// TwinCAT 3 PLC project Untitled1
// ProgramVersion: 3.1.4024.0
// libraries:
//   Tc2_Standard, * (Beckhoff Automation GmbH)
//   Tc2_System, * (Beckhoff Automation GmbH)
//   Tc3_Module, * (Beckhoff Automation GmbH)
//   VisuSymbols,3.5.10.0,System
// project tree:
//   / GlobalTextList.TcGTLO, PlcTask.TcTTO, Visualization Manager.TcVMO (not stored), Visualization.TcVIS
//   GVLs/ GVL.TcGVL
//   POUs/ MAIN.TcPOU, VeranderLicht.TcPOU, VerkeersLichtL.TcPOU, VerkeersLichtR.TcPOU, VerkeerslichtStatus.TcTLEO
// real-time tasks:
//   TASK PlcTask: cycle T#10ms, priority 20, ADS port 350
//   TASK Task 4: cycle T#10ms, priority 1, ADS port 351

CONFIGURATION Untitled1
    RESOURCE PLC ON TwinCAT3
        TASK PlcTask(INTERVAL := T#10ms, PRIORITY := 20);
        PROGRAM MAIN WITH PlcTask : MAIN;
    END_RESOURCE
END_CONFIGURATION

// ---- POUs/VerkeerslichtStatus.TcTLEO
{attribute 'qualified_only'}
{attribute 'strict'}
TYPE VerkeerslichtStatus :
(
	Rood := 0,    // 0
    Geel := 1,    // 1
    Groen := 2    // 2
);
END_TYPE

// ---- GVLs/GVL.TcGVL
{attribute 'qualified_only'}
VAR_GLOBAL
	GroenR : BOOL; 
	GeelR : BOOL;
	RoodR: BOOL;
	GroenL : BOOL;
	GeelL : BOOL;
	RoodL: BOOL;
	
	LichtStatusR: INT := 0; // 0 = Rood, 1 = Groen, 2 = Oranje
	LichtStatusL: INT := 0; // 0 = Rood, 1 = Groen, 2 = Oranje
	
	AutoR : BOOL; // Auto komt van Rechts
	AutoL : BOOL; // Auto komt van Links
	
	TijdGroen : TIME := T#5S; // de tijden zet ik hier neer zodat ik die makkelijk kan aanpassen
	TijdGeel : TIME := T#2S;
	TijdRood : TIME := T#5S;
	
END_VAR

// ---- POUs/MAIN.TcPOU
PROGRAM MAIN
VAR
	VeranderLicht: INT;
	StoplichtStatus: INT;
	StoplichtWissel: ENUM;
	Rood: INT;
	Groen: INT;
	Geel: INT;
	Entry1 : BOOL := TRUE;
END_VAR


IF  Entry1 THEN
    // Initialiseer alle verkeerslichtstatussen naar Rood
    GVL.LichtStatusR := Rood;
    GVL.LichtStatusL := Rood;
    Entry1 := FALSE;  // Voorkom dat de initialisatie elke cyclus herhaald wordt
END_IF;

VerkeerslichtR();
VerkeerslichtL();

END_PROGRAM

// ---- POUs/VeranderLicht.TcPOU
FUNCTION VeranderLicht : VerkeerslichtStatus
VAR_INPUT
	StoplichtWissel	: VerkeerslichtStatus;
END_VAR


CASE StoplichtWissel OF
    VerkeerslichtStatus.Rood:
        VeranderLicht := VerkeerslichtStatus.Groen;   // Van Rood naar Groen
		
    VerkeerslichtStatus.Groen:
        VeranderLicht := VerkeerslichtStatus.Geel;  // Van Groen naar Geel
		
    VerkeerslichtStatus.Geel:
        VeranderLicht := VerkeerslichtStatus.Rood;    // Van Geel naar Rood
		
ELSE
    VeranderLicht := VerkeerslichtStatus.Rood;      // bij default moet het naar Rood
END_CASE

END_FUNCTION

// ---- POUs/VerkeersLichtR.TcPOU
PROGRAM VerkeersLichtR
VAR
	HuidigeStatus : VerkeerslichtStatus := VerkeerslichtStatus.Rood; //Start met rood
    Timer1 : TON; 
END_VAR


IF GVL.AutoR THEN //Als er een auto bij het stoplicht staat (de knop naast de lichten)
    CASE HuidigeStatus OF
        VerkeerslichtStatus.Rood:
            Timer1(IN := TRUE, PT := GVL.TijdRood);
            IF Timer1.Q THEN
                HuidigeStatus := VeranderLicht(HuidigeStatus);
                Timer1(IN := FALSE);
				
				GVL.GroenR := FALSE;
            	GVL.GeelR := FALSE;
            	GVL.RoodR := TRUE;   // Zet Rood licht aan

            END_IF
        VerkeerslichtStatus.Groen:
            Timer1(IN := TRUE, PT := GVL.TijdGroen);
            IF Timer1.Q THEN
                HuidigeStatus := VeranderLicht(HuidigeStatus);
                Timer1(IN := FALSE);
				
				GVL.GroenR := TRUE;   // Zet Groen licht aan
            	GVL.GeelR := FALSE;
           		GVL.RoodR := FALSE;
				
            END_IF
        VerkeerslichtStatus.Geel:
            Timer1(IN := TRUE, PT := GVL.TijdGeel);
            IF Timer1.Q THEN
                HuidigeStatus := VeranderLicht(HuidigeStatus);
                Timer1(IN := FALSE);
				
				GVL.GroenR := FALSE;
           		GVL.GeelR := TRUE;    // Zet Geel licht aan
            	GVL.RoodR := FALSE;
            END_IF
    END_CASE
ELSE
    // Als er geen auto aankomt, gaat het verkeerslicht op rood
    HuidigeStatus := VerkeerslichtStatus.Rood;
    GVL.GroenR := FALSE;
    GVL.GeelR := FALSE;
    GVL.RoodR := TRUE;
END_IF

GVL.LichtStatusR := HuidigeStatus; // Dit zorgt ervoor dat de GVL wordt ge-update

END_PROGRAM

// ---- POUs/VerkeersLichtL.TcPOU
PROGRAM VerkeersLichtL
VAR
	HuidigeStatus : VerkeerslichtStatus := VerkeerslichtStatus.Rood; //Start met rood
    Timer2 : TON; 
END_VAR


IF GVL.AutoL THEN //Als er een auto bij het stoplicht staat (de knop naast de lichten)
    CASE HuidigeStatus OF
        VerkeerslichtStatus.Rood:
            Timer2(IN := TRUE, PT := GVL.TijdRood);
            IF Timer2.Q THEN
                HuidigeStatus := VeranderLicht(HuidigeStatus);
                Timer2(IN := FALSE);
				
				GVL.GroenL := FALSE;
            	GVL.GeelL := FALSE;
            	GVL.RoodL := TRUE;   // Zet Rood licht aan

            END_IF
        VerkeerslichtStatus.Groen:
            Timer2(IN := TRUE, PT := GVL.TijdGroen);
            IF Timer2.Q THEN
                HuidigeStatus := VeranderLicht(HuidigeStatus);
                Timer2(IN := FALSE);
				
				GVL.GroenL := TRUE;   // Zet Groen licht aan
            	GVL.GeelL := FALSE;
           		GVL.RoodL := FALSE;
				
            END_IF
        VerkeerslichtStatus.Geel:
            Timer2(IN := TRUE, PT := GVL.TijdGeel);
            IF Timer2.Q THEN
                HuidigeStatus := VeranderLicht(HuidigeStatus);
                Timer2(IN := FALSE);
				
				GVL.GroenL := FALSE;
           		GVL.GeelL := TRUE;    // Zet Geel licht aan
            	GVL.RoodL := FALSE;
            END_IF
    END_CASE
ELSE
    // Als er geen auto aankomt, gaat het verkeerslicht op rood
    HuidigeStatus := VerkeerslichtStatus.Rood;
    GVL.GroenL := FALSE;
    GVL.GeelL := FALSE;
    GVL.RoodL := TRUE;
END_IF

GVL.LichtStatusL := HuidigeStatus; // Dit zorgt ervoor dat de GVL wordt ge-update

END_PROGRAM

// ---- Visualization.TcVIS
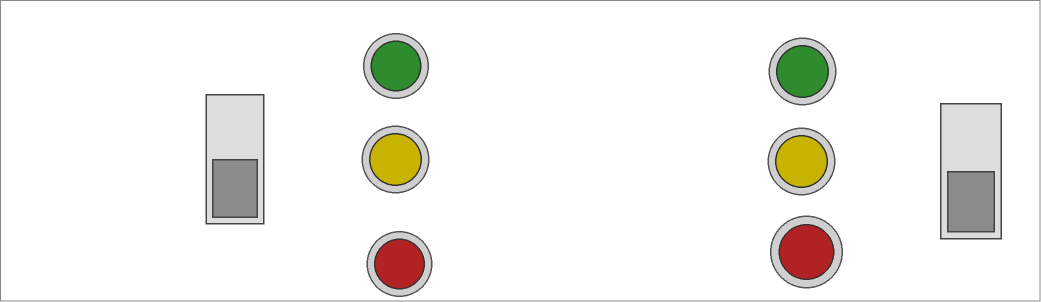
VISUALIZATION Visualization  // 1041x302
VAR
	//komt hier iets?
END_VAR
    Lamp1 (762,32 81x79), variable: GVL.GroenR, style: Lamp-Lamp1-Green
    Lamp1 (761,122 81x79), variable: GVL.GeelR, style: Lamp-Lamp1-Yellow
    Lamp1 (758,210 97x84), variable: GVL.RoodR, style: Lamp-Lamp1-Red
    Lamp1 (357,28 78x76), variable: GVL.GroenL, style: Lamp-Lamp1-Green
    Lamp1 (355,120 81x79), variable: GVL.GeelL, style: Lamp-Lamp1-Yellow
    Lamp1 (357,226 85x76), variable: GVL.RoodL, style: Lamp-Lamp1-Red
    DipSwitch (901,103 140x136), variable: GVL.AutoR, behaviour: TOGGLE, style: Switch-DipSwitch-Gray
    DipSwitch (167,94 136x130), variable: GVL.AutoL, behaviour: TOGGLE, style: Switch-DipSwitch-Gray
END_VISUALIZATION
